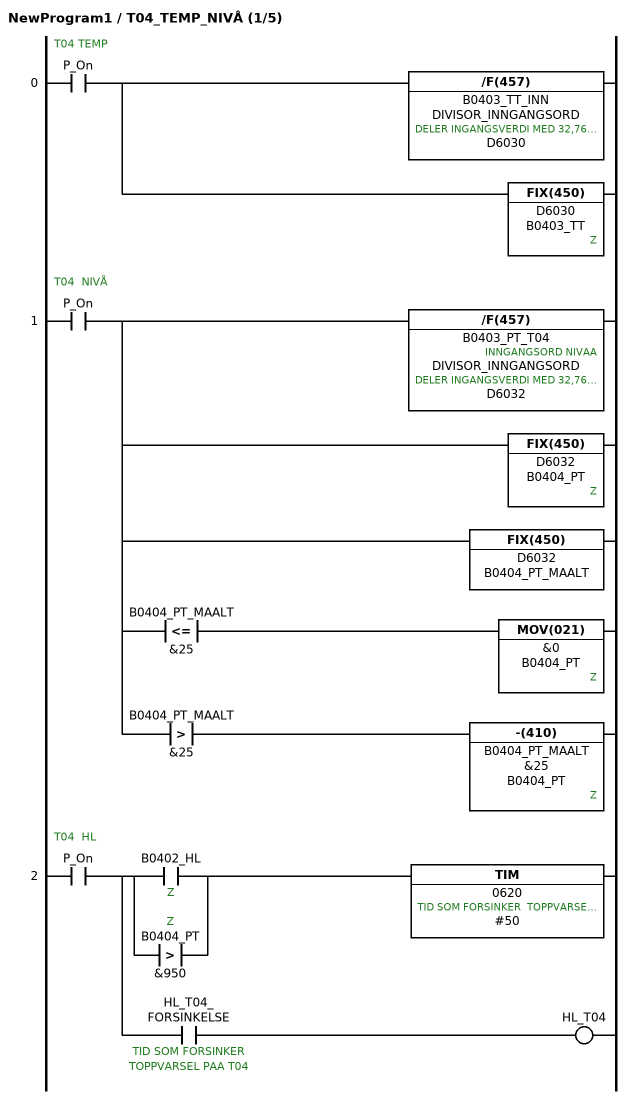
; [picture p912: NewProgram1 / T04_TEMP_NIVÅ, rungs 0-2]
; rung 0: T04 TEMP
LD P_On
/F(457) B0403_TT_INN DIVISOR_INNGANGSORD D6030  ; DELER INGANGSVERDI MED 32,760 FOR OMREGNING TIL 0-1000
FIX(450) D6030 B0403_TT  ; Z
; rung 1: T04  NIVÅ
LD P_On
OUT TR0
/F(457) B0403_PT_T04 DIVISOR_INNGANGSORD D6032  ; INNGANGSORD NIVAA, DELER INGANGSVERDI MED 32,760 FOR OMREGNING TIL 0-1000
FIX(450) D6032 B0404_PT  ; Z
FIX(450) D6032 B0404_PT_MAALT
AND<=(315) B0404_PT_MAALT &25
MOV(021) &0 B0404_PT  ; Z
LD TR0
AND>(320) B0404_PT_MAALT &25
-(410) B0404_PT_MAALT &25 B0404_PT  ; Z
; rung 2: T04  HL
LD P_On
OUT TR0
LD B0402_HL  ; Z
OR>(320) B0404_PT &950  ; Z
ANDLD
TIM 0620 #50  ; TID SOM FORSINKER  TOPPVARSEL PAA T04
LD TR0
AND HL_T04_FORSINKELSE  ; TID SOM FORSINKER  TOPPVARSEL PAA T04
OUT HL_T04

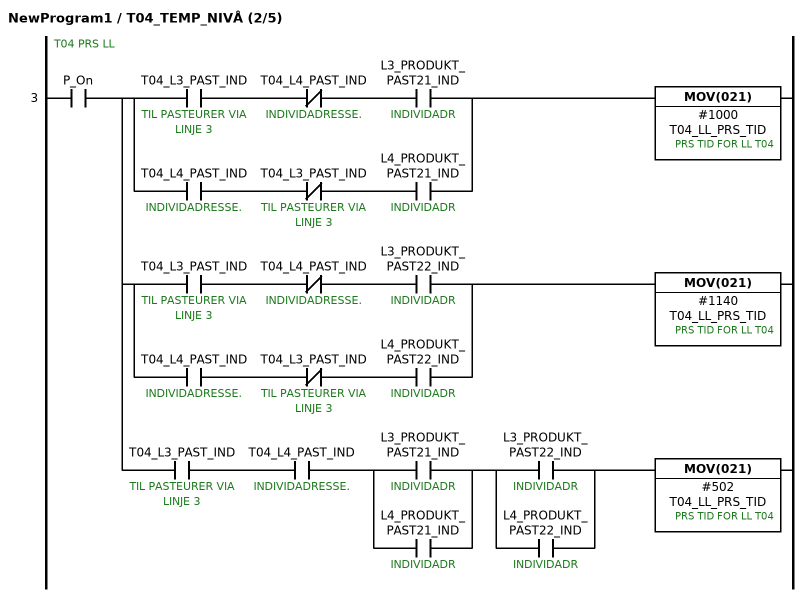
; rung 3: T04 PRS LL
LD P_On
OUT TR0
LD T04_L3_PAST_IND  ; TIL PASTEURER VIA LINJE 3
ANDNOT T04_L4_PAST_IND  ; INDIVIDADRESSE.
AND L3_PRODUKT_PAST21_IND  ; INDIVIDADR
LD T04_L4_PAST_IND  ; INDIVIDADRESSE.
ANDNOT T04_L3_PAST_IND  ; TIL PASTEURER VIA LINJE 3
AND L4_PRODUKT_PAST21_IND  ; INDIVIDADR
ORLD
ANDLD
MOV(021) #1000 T04_LL_PRS_TID  ; PRS TID FOR LL T04
LD TR0
LD T04_L3_PAST_IND  ; TIL PASTEURER VIA LINJE 3
ANDNOT T04_L4_PAST_IND  ; INDIVIDADRESSE.
AND L3_PRODUKT_PAST22_IND  ; INDIVIDADR
LD T04_L4_PAST_IND  ; INDIVIDADRESSE.
ANDNOT T04_L3_PAST_IND  ; TIL PASTEURER VIA LINJE 3
AND L4_PRODUKT_PAST22_IND  ; INDIVIDADR
ORLD
ANDLD
MOV(021) #1140 T04_LL_PRS_TID  ; PRS TID FOR LL T04
LD TR0
AND T04_L3_PAST_IND  ; TIL PASTEURER VIA LINJE 3
AND T04_L4_PAST_IND  ; INDIVIDADRESSE.
LD L3_PRODUKT_PAST21_IND  ; INDIVIDADR
OR L4_PRODUKT_PAST21_IND  ; INDIVIDADR
ANDLD
LD L3_PRODUKT_PAST22_IND  ; INDIVIDADR
OR L4_PRODUKT_PAST22_IND  ; INDIVIDADR
ANDLD
MOV(021) #502 T04_LL_PRS_TID  ; PRS TID FOR LL T04

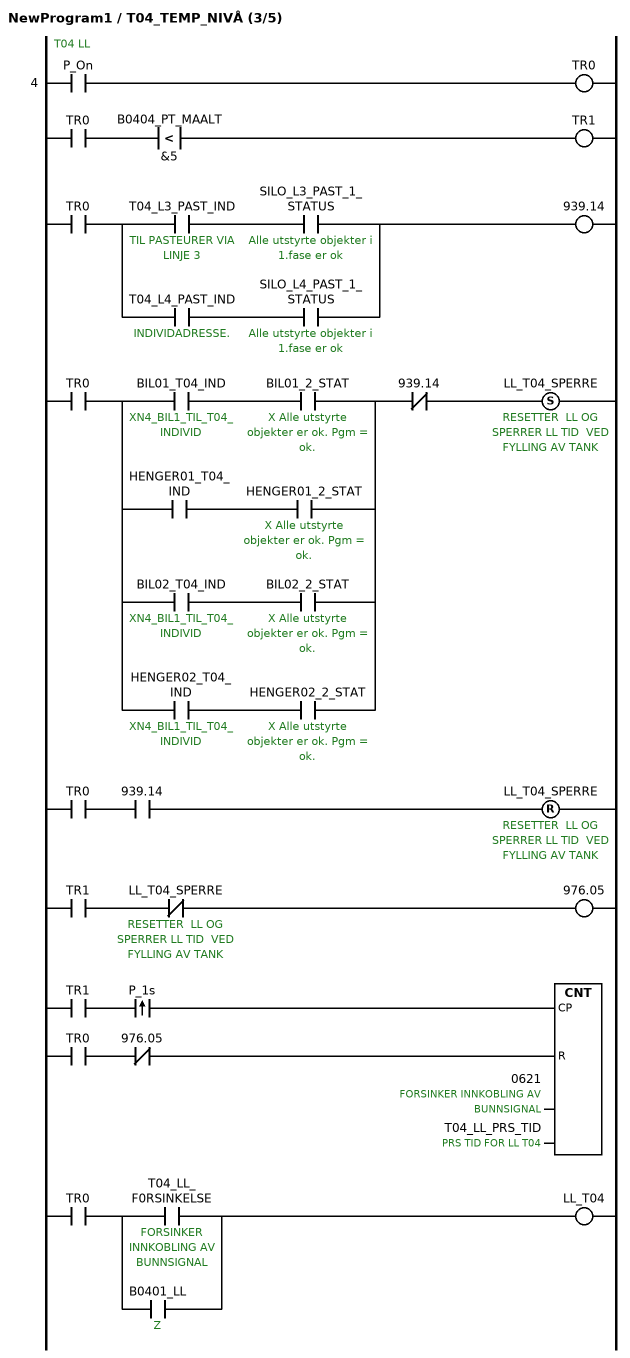
; rung 4: T04 LL
LD P_On
OUT TR0
LD T04_L3_PAST_IND  ; TIL PASTEURER VIA LINJE 3
AND SILO_L3_PAST_1_STATUS  ; Alle utstyrte objekter i 1.fase er ok
LD T04_L4_PAST_IND  ; INDIVIDADRESSE.
AND SILO_L4_PAST_1_STATUS  ; Alle utstyrte objekter i 1.fase er ok
ORLD
ANDLD
OUT 939.14
LD TR0
LD BIL01_T04_IND  ; XN4_BIL1_TIL_T04_INDIVID
AND BIL01_2_STAT  ; X Alle utstyrte objekter er ok. Pgm = ok.
LD HENGER01_T04_IND
AND HENGER01_2_STAT  ; X Alle utstyrte objekter er ok. Pgm = ok.
ORLD
LD BIL02_T04_IND  ; XN4_BIL1_TIL_T04_INDIVID
AND BIL02_2_STAT  ; X Alle utstyrte objekter er ok. Pgm = ok.
ORLD
LD HENGER02_T04_IND  ; XN4_BIL1_TIL_T04_INDIVID
AND HENGER02_2_STAT  ; X Alle utstyrte objekter er ok. Pgm = ok.
ORLD
ANDLD
ANDNOT 939.14
SET LL_T04_SPERRE  ; RESETTER  LL OG SPERRER LL TID  VED FYLLING AV TANK
LD TR0
AND 939.14
RSET LL_T04_SPERRE  ; RESETTER  LL OG SPERRER LL TID  VED FYLLING AV TANK
LD TR0
AND<(310) B0404_PT_MAALT &5
OUT TR1
ANDNOT LL_T04_SPERRE  ; RESETTER  LL OG SPERRER LL TID  VED FYLLING AV TANK
OUT 976.05
LD TR1
@AND P_1s
LD TR0
ANDNOT 976.05
CNT 0621 T04_LL_PRS_TID  ; PRS TID FOR LL T04, FORSINKER INNKOBLING AV BUNNSIGNAL
LD TR0
LD T04_LL_F0RSINKELSE  ; FORSINKER INNKOBLING AV BUNNSIGNAL
OR B0401_LL  ; Z
ANDLD
OUT LL_T04

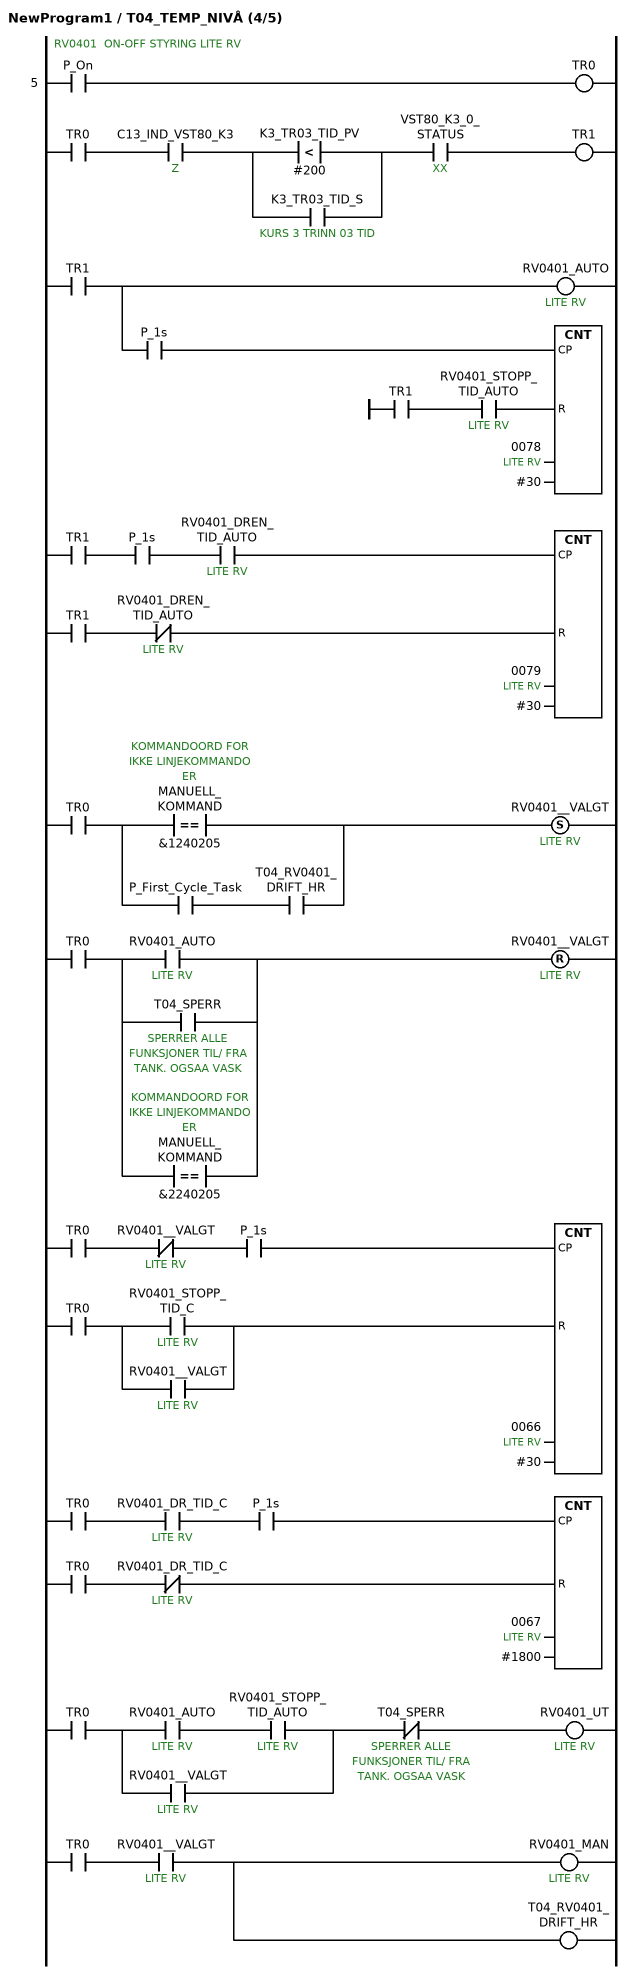
; rung 5: RV0401  ON-OFF STYRING LITE RV
LD P_On
OUT TR0
AND C13_IND_VST80_K3  ; Z
LD<(310) K3_TR03_TID_PV #200
OR K3_TR03_TID_S  ; KURS 3 TRINN 03 TID
ANDLD
AND VST80_K3_0_STATUS  ; XX
OUT TR1
OUT RV0401_AUTO  ; LITE RV
AND P_1s
LD TR1
AND RV0401_STOPP_TID_AUTO  ; LITE RV
CNT 0078 #30  ; LITE RV
LD TR1
AND P_1s
AND RV0401_DREN_TID_AUTO  ; LITE RV
LD TR1
ANDNOT RV0401_DREN_TID_AUTO  ; LITE RV
CNT 0079 #30  ; LITE RV
LD TR0
LD=L(301) MANUELL_KOMMAND &1240205  ; KOMMANDOORD FOR IKKE LINJEKOMMANDOER
LD P_First_Cycle_Task
AND T04_RV0401_DRIFT_HR
ORLD
ANDLD
SET RV0401__VALGT  ; LITE RV
LD TR0
LD RV0401_AUTO  ; LITE RV
OR T04_SPERR  ; SPERRER ALLE FUNKSJONER TIL/ FRA TANK. OGSAA VASK
OR=L(301) MANUELL_KOMMAND &2240205  ; KOMMANDOORD FOR IKKE LINJEKOMMANDOER
ANDLD
RSET RV0401__VALGT  ; LITE RV
LD TR0
ANDNOT RV0401__VALGT  ; LITE RV
AND P_1s
LD TR0
LD RV0401_STOPP_TID_C  ; LITE RV
OR RV0401__VALGT  ; LITE RV
ANDLD
CNT 0066 #30  ; LITE RV
LD TR0
AND RV0401_DR_TID_C  ; LITE RV
AND P_1s
LD TR0
ANDNOT RV0401_DR_TID_C  ; LITE RV
CNT 0067 #1800  ; LITE RV
LD TR0
LD RV0401_AUTO  ; LITE RV
AND RV0401_STOPP_TID_AUTO  ; LITE RV
OR RV0401__VALGT  ; LITE RV
ANDLD
ANDNOT T04_SPERR  ; SPERRER ALLE FUNKSJONER TIL/ FRA TANK. OGSAA VASK
OUT RV0401_UT  ; LITE RV
LD TR0
AND RV0401__VALGT  ; LITE RV
OUT RV0401_MAN  ; LITE RV
OUT T04_RV0401_DRIFT_HR

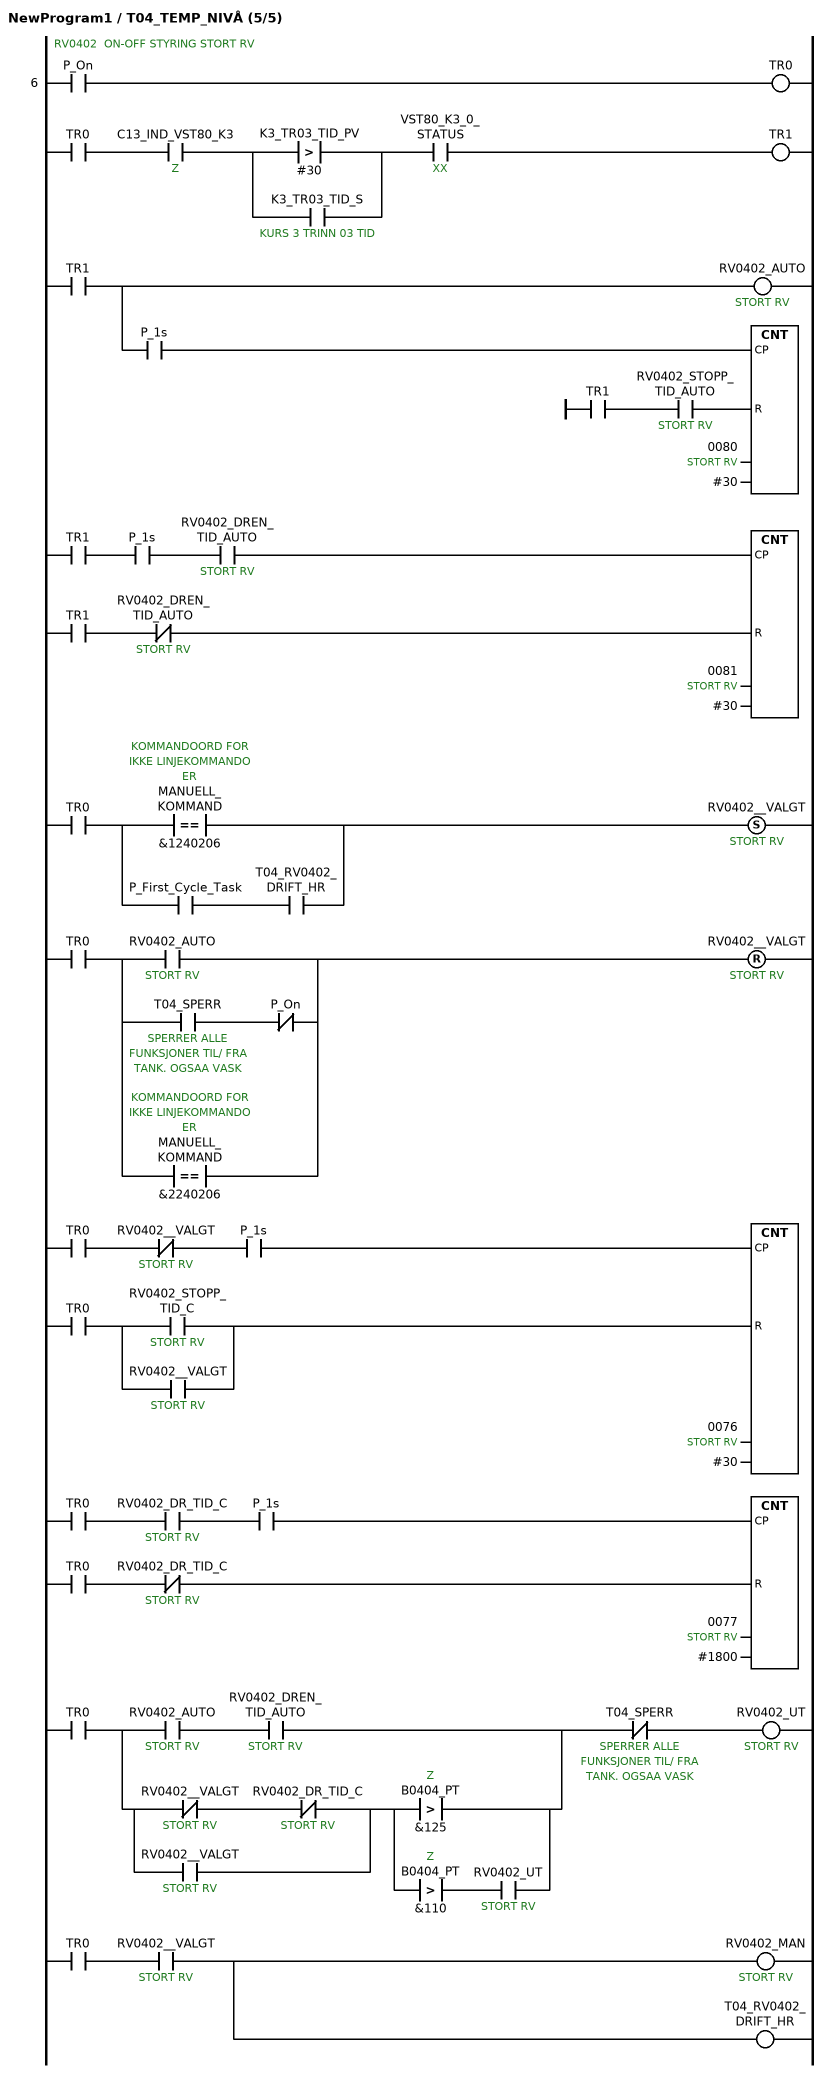
; rung 6: RV0402  ON-OFF STYRING STORT RV
LD P_On
OUT TR0
AND C13_IND_VST80_K3  ; Z
LD>(320) K3_TR03_TID_PV #30
OR K3_TR03_TID_S  ; KURS 3 TRINN 03 TID
ANDLD
AND VST80_K3_0_STATUS  ; XX
OUT TR1
OUT RV0402_AUTO  ; STORT RV
AND P_1s
LD TR1
AND RV0402_STOPP_TID_AUTO  ; STORT RV
CNT 0080 #30  ; STORT RV
LD TR1
AND P_1s
AND RV0402_DREN_TID_AUTO  ; STORT RV
LD TR1
ANDNOT RV0402_DREN_TID_AUTO  ; STORT RV
CNT 0081 #30  ; STORT RV
LD TR0
LD=L(301) MANUELL_KOMMAND &1240206  ; KOMMANDOORD FOR IKKE LINJEKOMMANDOER
LD P_First_Cycle_Task
AND T04_RV0402_DRIFT_HR
ORLD
ANDLD
SET RV0402__VALGT  ; STORT RV
LD TR0
LD RV0402_AUTO  ; STORT RV
LD T04_SPERR  ; SPERRER ALLE FUNKSJONER TIL/ FRA TANK. OGSAA VASK
ANDNOT P_On
ORLD
OR=L(301) MANUELL_KOMMAND &2240206  ; KOMMANDOORD FOR IKKE LINJEKOMMANDOER
ANDLD
RSET RV0402__VALGT  ; STORT RV
LD TR0
ANDNOT RV0402__VALGT  ; STORT RV
AND P_1s
LD TR0
LD RV0402_STOPP_TID_C  ; STORT RV
OR RV0402__VALGT  ; STORT RV
ANDLD
CNT 0076 #30  ; STORT RV
LD TR0
AND RV0402_DR_TID_C  ; STORT RV
AND P_1s
LD TR0
ANDNOT RV0402_DR_TID_C  ; STORT RV
CNT 0077 #1800  ; STORT RV
LD TR0
LD RV0402_AUTO  ; STORT RV
AND RV0402_DREN_TID_AUTO  ; STORT RV
LDNOT RV0402__VALGT  ; STORT RV
ANDNOT RV0402_DR_TID_C  ; STORT RV
OR RV0402__VALGT  ; STORT RV
LD>(320) B0404_PT &125  ; Z
LD>(320) B0404_PT &110  ; Z
AND RV0402_UT  ; STORT RV
ORLD
ANDLD
ORLD
ANDLD
ANDNOT T04_SPERR  ; SPERRER ALLE FUNKSJONER TIL/ FRA TANK. OGSAA VASK
OUT RV0402_UT  ; STORT RV
LD TR0
AND RV0402__VALGT  ; STORT RV
OUT RV0402_MAN  ; STORT RV
OUT T04_RV0402_DRIFT_HR
; rung 7: Ingen_kommentar_funnet

### Section T04_STATUS

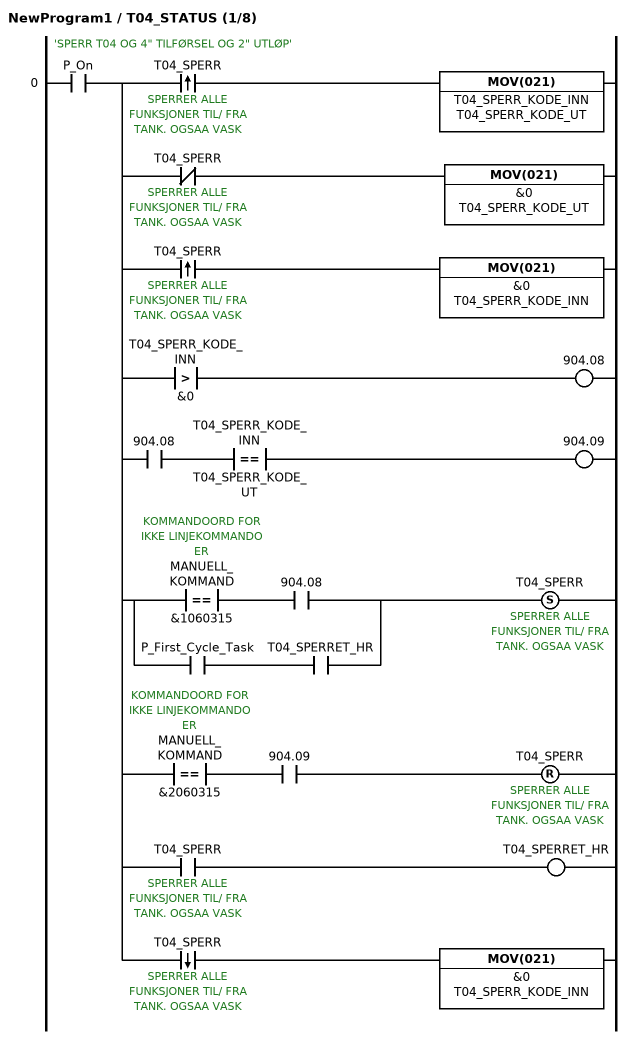
; rung 0: 'SPERR T04 OG 4" TILFØRSEL OG 2" UTLØP'
LD P_On
OUT TR0
@AND T04_SPERR  ; SPERRER ALLE FUNKSJONER TIL/ FRA TANK. OGSAA VASK
MOV(021) T04_SPERR_KODE_INN T04_SPERR_KODE_UT
LD TR0
ANDNOT T04_SPERR  ; SPERRER ALLE FUNKSJONER TIL/ FRA TANK. OGSAA VASK
MOV(021) &0 T04_SPERR_KODE_UT
LD TR0
@AND T04_SPERR  ; SPERRER ALLE FUNKSJONER TIL/ FRA TANK. OGSAA VASK
MOV(021) &0 T04_SPERR_KODE_INN
LD TR0
AND>(320) T04_SPERR_KODE_INN &0
OUT 904.08
LD TR0
AND 904.08
AND=(300) T04_SPERR_KODE_INN T04_SPERR_KODE_UT
OUT 904.09
LD TR0
LD=L(301) MANUELL_KOMMAND &1060315  ; KOMMANDOORD FOR IKKE LINJEKOMMANDOER
AND 904.08
LD P_First_Cycle_Task
AND T04_SPERRET_HR
ORLD
ANDLD
SET T04_SPERR  ; SPERRER ALLE FUNKSJONER TIL/ FRA TANK. OGSAA VASK
LD TR0
AND=L(301) MANUELL_KOMMAND &2060315  ; KOMMANDOORD FOR IKKE LINJEKOMMANDOER
AND 904.09
RSET T04_SPERR  ; SPERRER ALLE FUNKSJONER TIL/ FRA TANK. OGSAA VASK
LD TR0
AND T04_SPERR  ; SPERRER ALLE FUNKSJONER TIL/ FRA TANK. OGSAA VASK
OUT T04_SPERRET_HR
LD TR0
%AND T04_SPERR  ; SPERRER ALLE FUNKSJONER TIL/ FRA TANK. OGSAA VASK
MOV(021) &0 T04_SPERR_KODE_INN

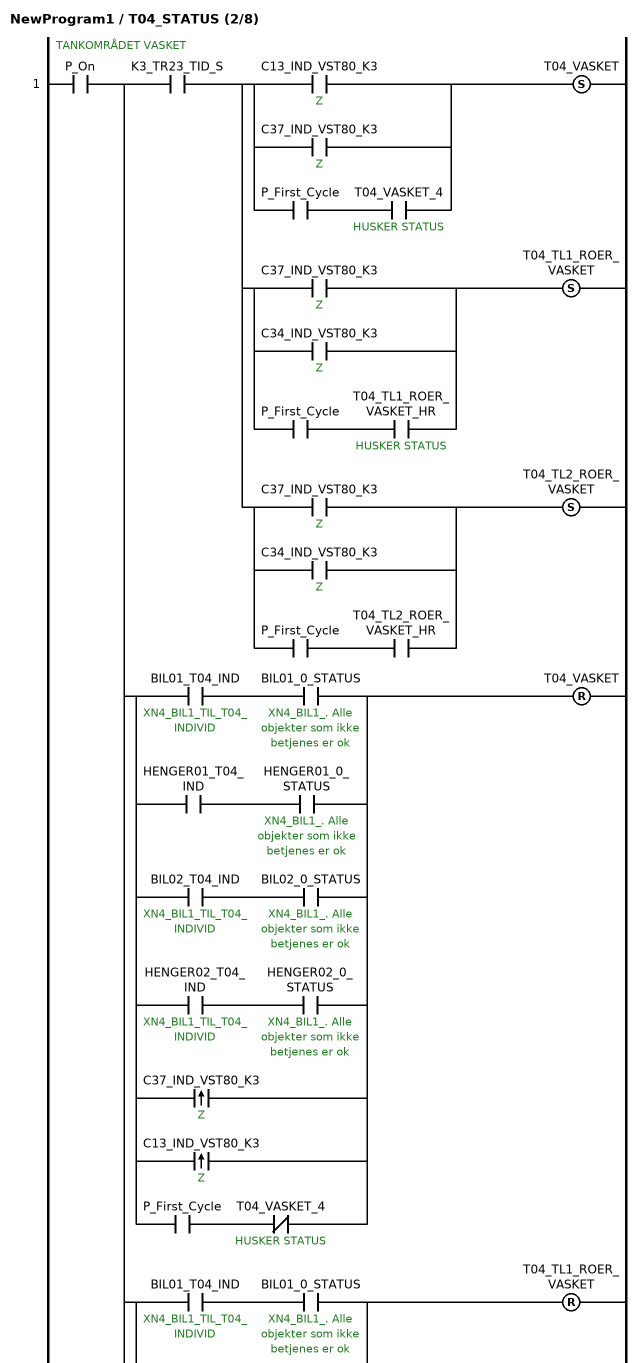

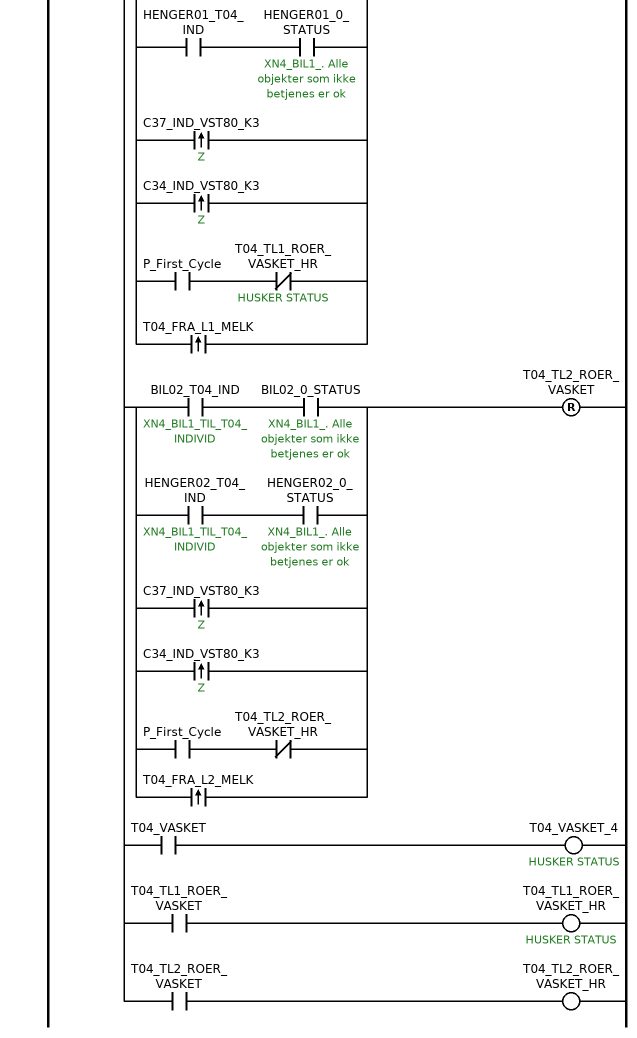
; rung 1: TANKOMRÅDET VASKET
LD P_On
OUT TR0
AND K3_TR23_TID_S
OUT TR1
LD C13_IND_VST80_K3  ; Z
OR C37_IND_VST80_K3  ; Z
LD P_First_Cycle
AND T04_VASKET_4  ; HUSKER STATUS
ORLD
ANDLD
SET T04_VASKET
LD TR1
LD C37_IND_VST80_K3  ; Z
OR C34_IND_VST80_K3  ; Z
LD P_First_Cycle
AND T04_TL1_ROER_VASKET_HR  ; HUSKER STATUS
ORLD
ANDLD
SET T04_TL1_ROER_VASKET
LD TR1
LD C37_IND_VST80_K3  ; Z
OR C34_IND_VST80_K3  ; Z
LD P_First_Cycle
AND T04_TL2_ROER_VASKET_HR
ORLD
ANDLD
SET T04_TL2_ROER_VASKET
LD TR0
LD BIL01_T04_IND  ; XN4_BIL1_TIL_T04_INDIVID
AND BIL01_0_STATUS  ; XN4_BIL1_. Alle objekter som ikke betjenes er ok
LD HENGER01_T04_IND
AND HENGER01_0_STATUS  ; XN4_BIL1_. Alle objekter som ikke betjenes er ok
ORLD
LD BIL02_T04_IND  ; XN4_BIL1_TIL_T04_INDIVID
AND BIL02_0_STATUS  ; XN4_BIL1_. Alle objekter som ikke betjenes er ok
ORLD
LD HENGER02_T04_IND  ; XN4_BIL1_TIL_T04_INDIVID
AND HENGER02_0_STATUS  ; XN4_BIL1_. Alle objekter som ikke betjenes er ok
ORLD
@OR C37_IND_VST80_K3  ; Z
@OR C13_IND_VST80_K3  ; Z
LD P_First_Cycle
ANDNOT T04_VASKET_4  ; HUSKER STATUS
ORLD
ANDLD
RSET T04_VASKET
LD TR0
LD BIL01_T04_IND  ; XN4_BIL1_TIL_T04_INDIVID
AND BIL01_0_STATUS  ; XN4_BIL1_. Alle objekter som ikke betjenes er ok
LD HENGER01_T04_IND
AND HENGER01_0_STATUS  ; XN4_BIL1_. Alle objekter som ikke betjenes er ok
ORLD
@OR C37_IND_VST80_K3  ; Z
@OR C34_IND_VST80_K3  ; Z
LD P_First_Cycle
ANDNOT T04_TL1_ROER_VASKET_HR  ; HUSKER STATUS
ORLD
@OR T04_FRA_L1_MELK
ANDLD
RSET T04_TL1_ROER_VASKET
LD TR0
LD BIL02_T04_IND  ; XN4_BIL1_TIL_T04_INDIVID
AND BIL02_0_STATUS  ; XN4_BIL1_. Alle objekter som ikke betjenes er ok
LD HENGER02_T04_IND  ; XN4_BIL1_TIL_T04_INDIVID
AND HENGER02_0_STATUS  ; XN4_BIL1_. Alle objekter som ikke betjenes er ok
ORLD
@OR C37_IND_VST80_K3  ; Z
@OR C34_IND_VST80_K3  ; Z
LD P_First_Cycle
ANDNOT T04_TL2_ROER_VASKET_HR
ORLD
@OR T04_FRA_L2_MELK
ANDLD
RSET T04_TL2_ROER_VASKET
LD TR0
AND T04_VASKET
OUT T04_VASKET_4  ; HUSKER STATUS
LD TR0
AND T04_TL1_ROER_VASKET
OUT T04_TL1_ROER_VASKET_HR  ; HUSKER STATUS
LD TR0
AND T04_TL2_ROER_VASKET
OUT T04_TL2_ROER_VASKET_HR

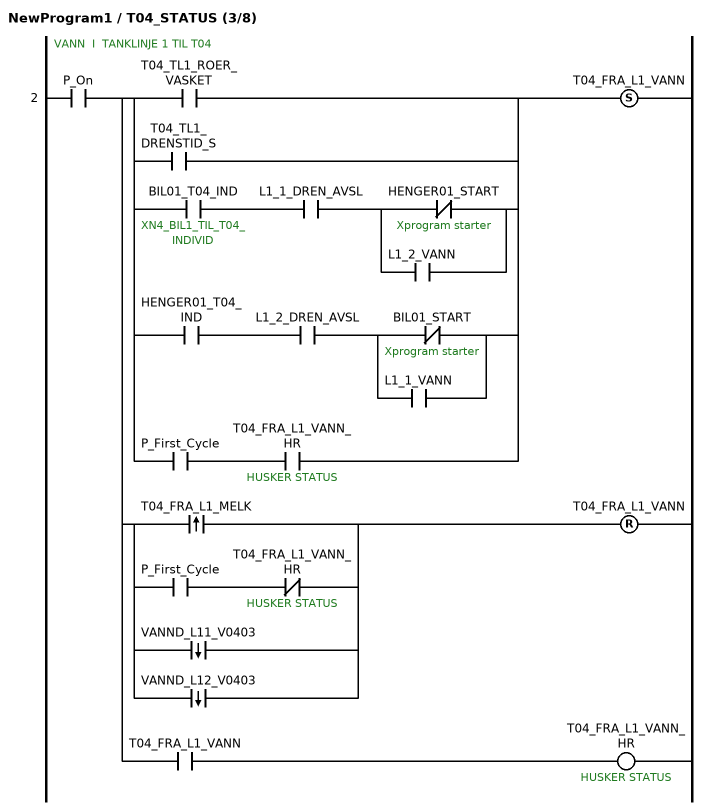
; rung 2: VANN  I  TANKLINJE 1 TIL T04
LD P_On
OUT TR0
LD T04_TL1_ROER_VASKET
OR T04_TL1_DRENSTID_S
LD BIL01_T04_IND  ; XN4_BIL1_TIL_T04_INDIVID
AND L1_1_DREN_AVSL
LDNOT HENGER01_START  ; Xprogram starter
OR L1_2_VANN
ANDLD
ORLD
LD HENGER01_T04_IND
AND L1_2_DREN_AVSL
LDNOT BIL01_START  ; Xprogram starter
OR L1_1_VANN
ANDLD
ORLD
LD P_First_Cycle
AND T04_FRA_L1_VANN_HR  ; HUSKER STATUS
ORLD
ANDLD
SET T04_FRA_L1_VANN
LD TR0
@LD T04_FRA_L1_MELK
LD P_First_Cycle
ANDNOT T04_FRA_L1_VANN_HR  ; HUSKER STATUS
ORLD
%OR VANND_L11_V0403
%OR VANND_L12_V0403
ANDLD
RSET T04_FRA_L1_VANN
LD TR0
AND T04_FRA_L1_VANN
OUT T04_FRA_L1_VANN_HR  ; HUSKER STATUS

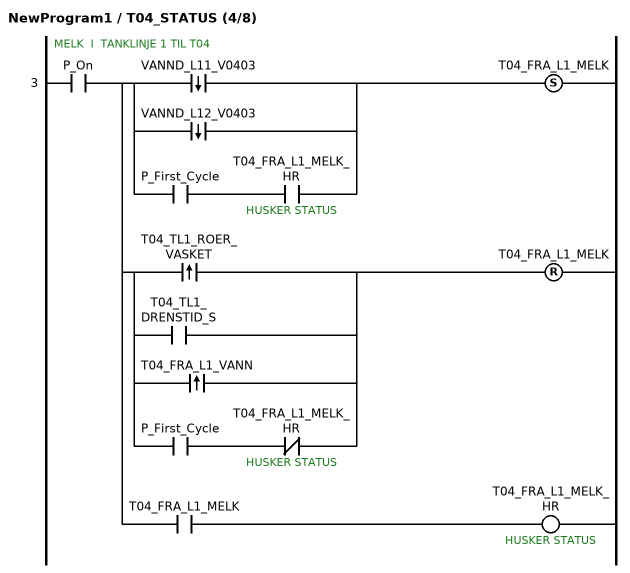
; rung 3: MELK  I  TANKLINJE 1 TIL T04
LD P_On
OUT TR0
%LD VANND_L11_V0403
%OR VANND_L12_V0403
LD P_First_Cycle
AND T04_FRA_L1_MELK_HR  ; HUSKER STATUS
ORLD
ANDLD
SET T04_FRA_L1_MELK
LD TR0
@LD T04_TL1_ROER_VASKET
OR T04_TL1_DRENSTID_S
@OR T04_FRA_L1_VANN
LD P_First_Cycle
ANDNOT T04_FRA_L1_MELK_HR  ; HUSKER STATUS
ORLD
ANDLD
RSET T04_FRA_L1_MELK
LD TR0
AND T04_FRA_L1_MELK
OUT T04_FRA_L1_MELK_HR  ; HUSKER STATUS

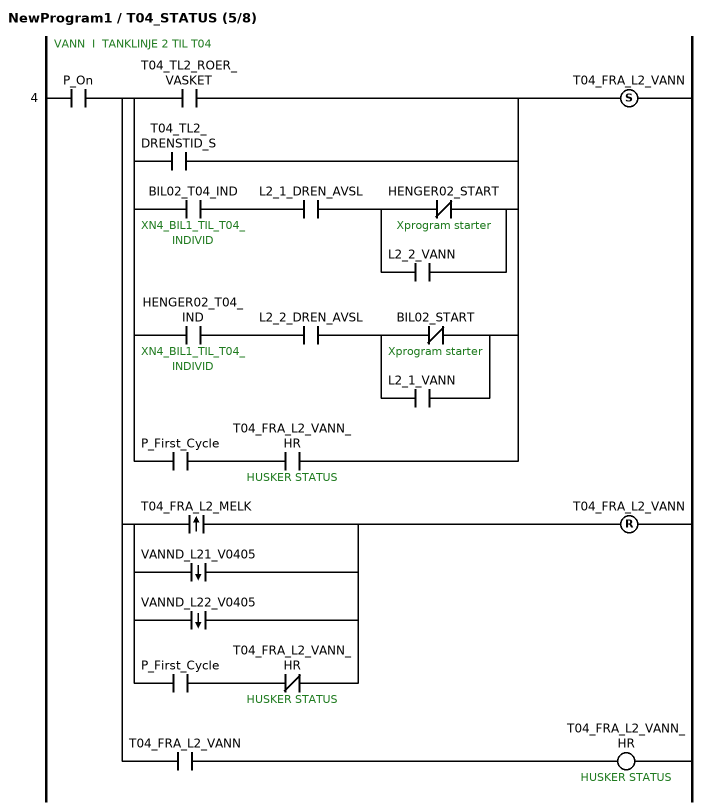
; rung 4: VANN  I  TANKLINJE 2 TIL T04
LD P_On
OUT TR0
LD T04_TL2_ROER_VASKET
OR T04_TL2_DRENSTID_S
LD BIL02_T04_IND  ; XN4_BIL1_TIL_T04_INDIVID
AND L2_1_DREN_AVSL
LDNOT HENGER02_START  ; Xprogram starter
OR L2_2_VANN
ANDLD
ORLD
LD HENGER02_T04_IND  ; XN4_BIL1_TIL_T04_INDIVID
AND L2_2_DREN_AVSL
LDNOT BIL02_START  ; Xprogram starter
OR L2_1_VANN
ANDLD
ORLD
LD P_First_Cycle
AND T04_FRA_L2_VANN_HR  ; HUSKER STATUS
ORLD
ANDLD
SET T04_FRA_L2_VANN
LD TR0
@LD T04_FRA_L2_MELK
%OR VANND_L21_V0405
%OR VANND_L22_V0405
LD P_First_Cycle
ANDNOT T04_FRA_L2_VANN_HR  ; HUSKER STATUS
ORLD
ANDLD
RSET T04_FRA_L2_VANN
LD TR0
AND T04_FRA_L2_VANN
OUT T04_FRA_L2_VANN_HR  ; HUSKER STATUS

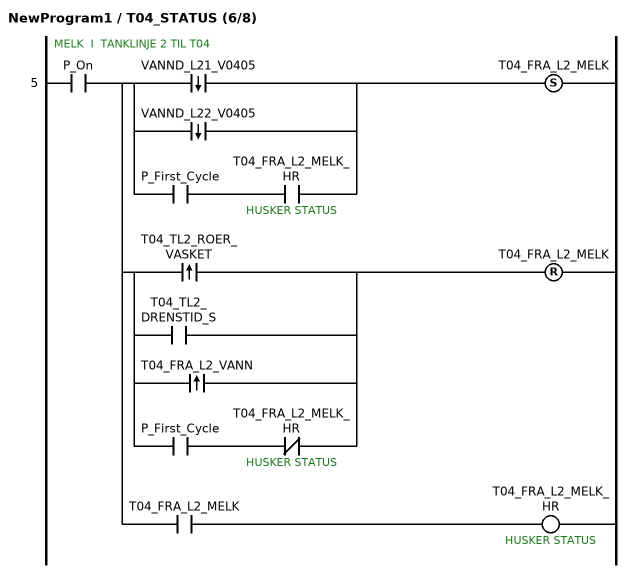
; rung 5: MELK  I  TANKLINJE 2 TIL T04
LD P_On
OUT TR0
%LD VANND_L21_V0405
%OR VANND_L22_V0405
LD P_First_Cycle
AND T04_FRA_L2_MELK_HR  ; HUSKER STATUS
ORLD
ANDLD
SET T04_FRA_L2_MELK
LD TR0
@LD T04_TL2_ROER_VASKET
OR T04_TL2_DRENSTID_S
@OR T04_FRA_L2_VANN
LD P_First_Cycle
ANDNOT T04_FRA_L2_MELK_HR  ; HUSKER STATUS
ORLD
ANDLD
RSET T04_FRA_L2_MELK
LD TR0
AND T04_FRA_L2_MELK
OUT T04_FRA_L2_MELK_HR  ; HUSKER STATUS

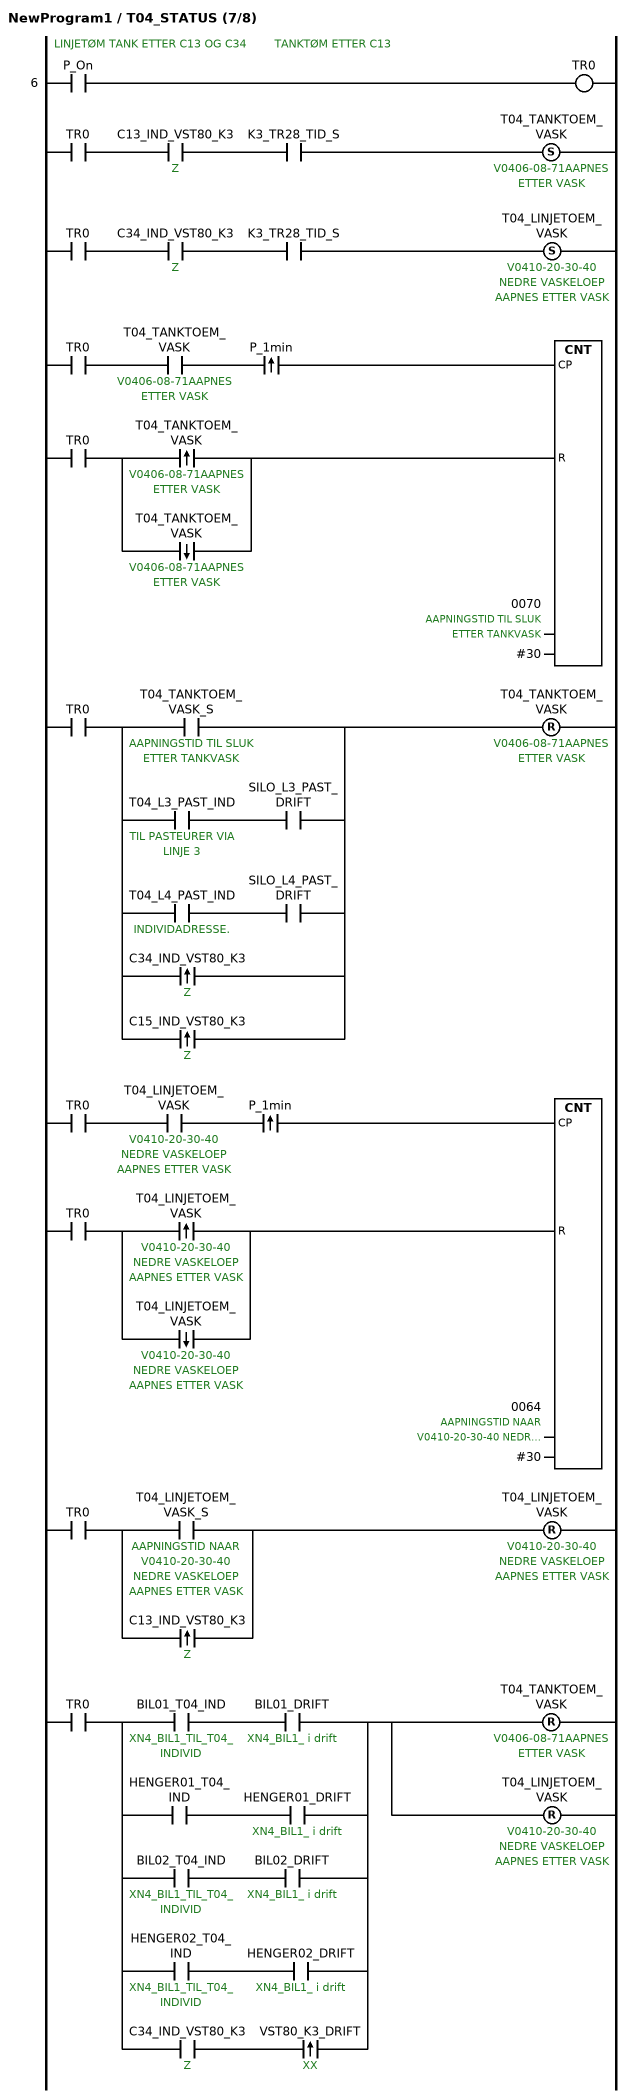
; rung 6: LINJETØM TANK ETTER C13 OG C34        TANKTØM ETTER C13
LD P_On
OUT TR0
AND C13_IND_VST80_K3  ; Z
AND K3_TR28_TID_S
SET T04_TANKTOEM_VASK  ; V0406-08-71AAPNES ETTER VASK
LD TR0
AND C34_IND_VST80_K3  ; Z
AND K3_TR28_TID_S
SET T04_LINJETOEM_VASK  ; V0410-20-30-40 NEDRE VASKELOEP AAPNES ETTER VASK
LD TR0
AND T04_TANKTOEM_VASK  ; V0406-08-71AAPNES ETTER VASK
@AND P_1min
LD TR0
@LD T04_TANKTOEM_VASK  ; V0406-08-71AAPNES ETTER VASK
%OR T04_TANKTOEM_VASK  ; V0406-08-71AAPNES ETTER VASK
ANDLD
CNT 0070 #30  ; AAPNINGSTID TIL SLUK ETTER TANKVASK
LD TR0
LD T04_TANKTOEM_VASK_S  ; AAPNINGSTID TIL SLUK ETTER TANKVASK
LD T04_L3_PAST_IND  ; TIL PASTEURER VIA LINJE 3
AND SILO_L3_PAST_DRIFT
ORLD
LD T04_L4_PAST_IND  ; INDIVIDADRESSE.
AND SILO_L4_PAST_DRIFT
ORLD
@OR C34_IND_VST80_K3  ; Z
@OR C15_IND_VST80_K3  ; Z
ANDLD
RSET T04_TANKTOEM_VASK  ; V0406-08-71AAPNES ETTER VASK
LD TR0
AND T04_LINJETOEM_VASK  ; V0410-20-30-40 NEDRE VASKELOEP AAPNES ETTER VASK
@AND P_1min
LD TR0
@LD T04_LINJETOEM_VASK  ; V0410-20-30-40 NEDRE VASKELOEP AAPNES ETTER VASK
%OR T04_LINJETOEM_VASK  ; V0410-20-30-40 NEDRE VASKELOEP AAPNES ETTER VASK
ANDLD
CNT 0064 #30  ; AAPNINGSTID NAAR V0410-20-30-40 NEDRE VASKELOEP AAPNES ETTER VASK
LD TR0
LD T04_LINJETOEM_VASK_S  ; AAPNINGSTID NAAR V0410-20-30-40 NEDRE VASKELOEP AAPNES ETTER VASK
@OR C13_IND_VST80_K3  ; Z
ANDLD
RSET T04_LINJETOEM_VASK  ; V0410-20-30-40 NEDRE VASKELOEP AAPNES ETTER VASK
LD TR0
LD BIL01_T04_IND  ; XN4_BIL1_TIL_T04_INDIVID
AND BIL01_DRIFT  ; XN4_BIL1_ i drift
LD HENGER01_T04_IND
AND HENGER01_DRIFT  ; XN4_BIL1_ i drift
ORLD
LD BIL02_T04_IND  ; XN4_BIL1_TIL_T04_INDIVID
AND BIL02_DRIFT  ; XN4_BIL1_ i drift
ORLD
LD HENGER02_T04_IND  ; XN4_BIL1_TIL_T04_INDIVID
AND HENGER02_DRIFT  ; XN4_BIL1_ i drift
ORLD
LD C34_IND_VST80_K3  ; Z
@AND VST80_K3_DRIFT  ; XX
ORLD
ANDLD
RSET T04_TANKTOEM_VASK  ; V0406-08-71AAPNES ETTER VASK
RSET T04_LINJETOEM_VASK  ; V0410-20-30-40 NEDRE VASKELOEP AAPNES ETTER VASK

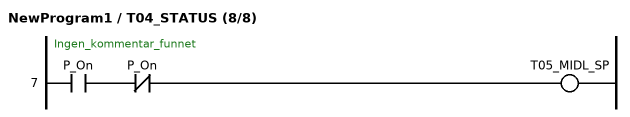
; rung 7: Ingen_kommentar_funnet
LD P_On
ANDNOT P_On
OUT T05_MIDL_SP
; rung 8: Ingen_kommentar_funnet

### Section T05_LOKALDREN

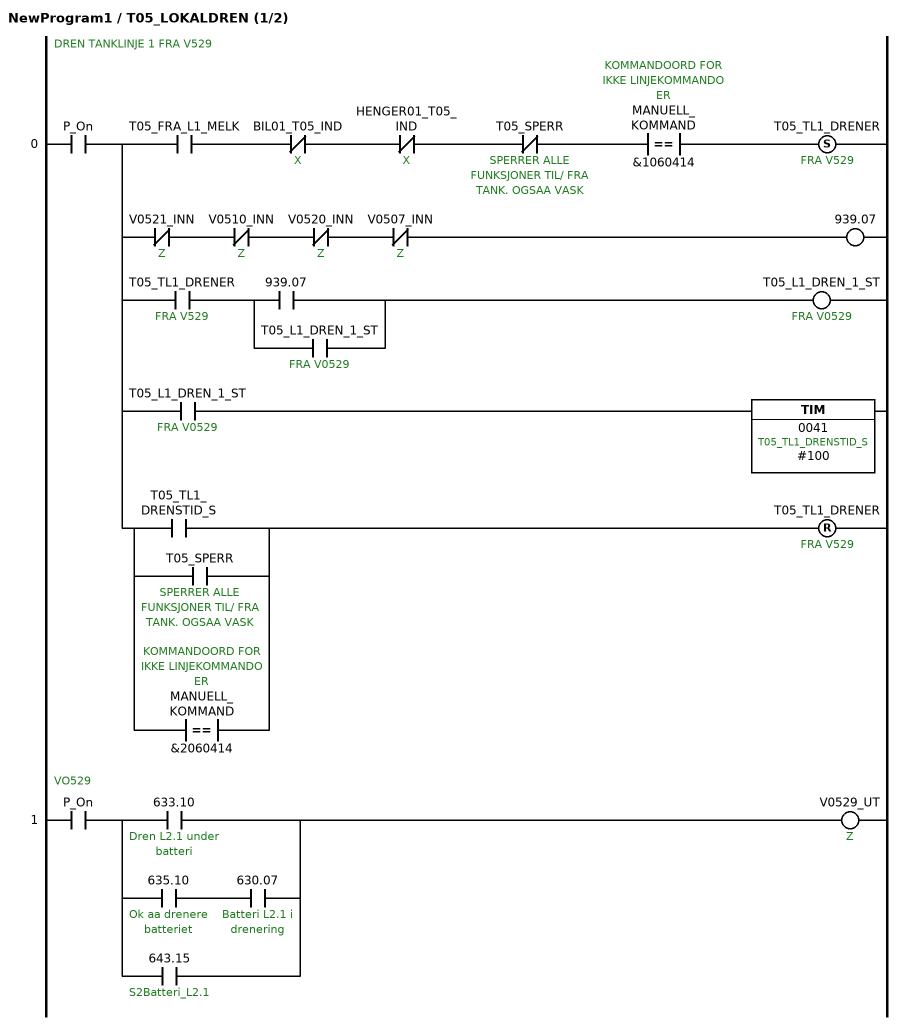
; rung 0: DREN TANKLINJE 1 FRA V529
LD P_On
OUT TR0
AND T05_FRA_L1_MELK
ANDNOT BIL01_T05_IND  ; X
ANDNOT HENGER01_T05_IND  ; X
ANDNOT T05_SPERR  ; SPERRER ALLE FUNKSJONER TIL/ FRA TANK. OGSAA VASK
AND=L(301) MANUELL_KOMMAND &1060414  ; KOMMANDOORD FOR IKKE LINJEKOMMANDOER
SET T05_TL1_DRENER  ; FRA V529
LD TR0
ANDNOT V0521_INN  ; Z
ANDNOT V0510_INN  ; Z
ANDNOT V0520_INN  ; Z
ANDNOT V0507_INN  ; Z
OUT 939.07
LD TR0
AND T05_TL1_DRENER  ; FRA V529
LD 939.07
OR T05_L1_DREN_1_ST  ; FRA V0529
ANDLD
OUT T05_L1_DREN_1_ST  ; FRA V0529
LD TR0
AND T05_L1_DREN_1_ST  ; FRA V0529
TIM 0041 #100  ; T05_TL1_DRENSTID_S
LD TR0
LD T05_TL1_DRENSTID_S
OR T05_SPERR  ; SPERRER ALLE FUNKSJONER TIL/ FRA TANK. OGSAA VASK
OR=L(301) MANUELL_KOMMAND &2060414  ; KOMMANDOORD FOR IKKE LINJEKOMMANDOER
ANDLD
RSET T05_TL1_DRENER  ; FRA V529
; rung 1: VO529
LD P_On
LD 633.10  ; Dren L2.1 under batteri
LD 635.10  ; Ok aa drenere batteriet
AND 630.07  ; Batteri L2.1 i drenering
ORLD
OR 643.15  ; S2Batteri_L2.1
ANDLD
OUT V0529_UT  ; Z

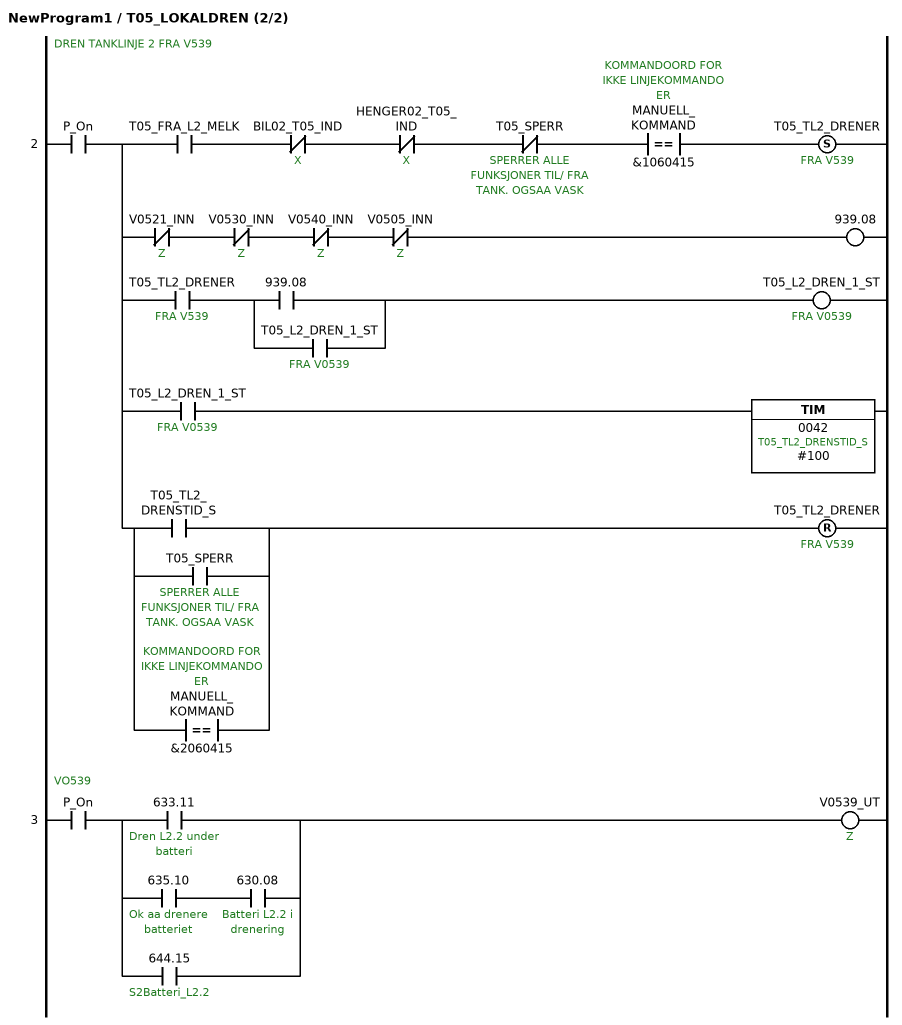
; rung 2: DREN TANKLINJE 2 FRA V539
LD P_On
OUT TR0
AND T05_FRA_L2_MELK
ANDNOT BIL02_T05_IND  ; X
ANDNOT HENGER02_T05_IND  ; X
ANDNOT T05_SPERR  ; SPERRER ALLE FUNKSJONER TIL/ FRA TANK. OGSAA VASK
AND=L(301) MANUELL_KOMMAND &1060415  ; KOMMANDOORD FOR IKKE LINJEKOMMANDOER
SET T05_TL2_DRENER  ; FRA V539
LD TR0
ANDNOT V0521_INN  ; Z
ANDNOT V0530_INN  ; Z
ANDNOT V0540_INN  ; Z
ANDNOT V0505_INN  ; Z
OUT 939.08
LD TR0
AND T05_TL2_DRENER  ; FRA V539
LD 939.08
OR T05_L2_DREN_1_ST  ; FRA V0539
ANDLD
OUT T05_L2_DREN_1_ST  ; FRA V0539
LD TR0
AND T05_L2_DREN_1_ST  ; FRA V0539
TIM 0042 #100  ; T05_TL2_DRENSTID_S
LD TR0
LD T05_TL2_DRENSTID_S
OR T05_SPERR  ; SPERRER ALLE FUNKSJONER TIL/ FRA TANK. OGSAA VASK
OR=L(301) MANUELL_KOMMAND &2060415  ; KOMMANDOORD FOR IKKE LINJEKOMMANDOER
ANDLD
RSET T05_TL2_DRENER  ; FRA V539
; rung 3: VO539
LD P_On
LD 633.11  ; Dren L2.2 under batteri
LD 635.10  ; Ok aa drenere batteriet
AND 630.08  ; Batteri L2.2 i drenering
ORLD
OR 644.15  ; S2Batteri_L2.2
ANDLD
OUT V0539_UT  ; Z
; rung 4: Ingen_kommentar_funnet

### Section T05_TEMP_NIVÅ

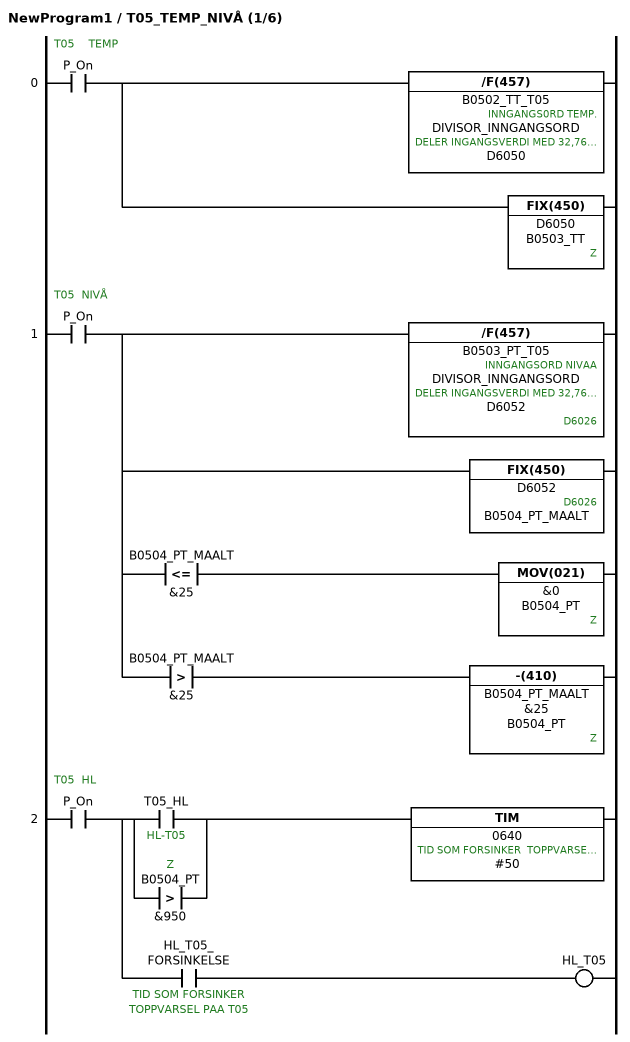
; rung 0: T05    TEMP
LD P_On
/F(457) B0502_TT_T05 DIVISOR_INNGANGSORD D6050  ; INNGANGS0RD TEMP., DELER INGANGSVERDI MED 32,760 FOR OMREGNING TIL 0-1000
FIX(450) D6050 B0503_TT  ; Z
; rung 1: T05  NIVÅ
LD P_On
OUT TR0
/F(457) B0503_PT_T05 DIVISOR_INNGANGSORD D6052  ; INNGANGSORD NIVAA, DELER INGANGSVERDI MED 32,760 FOR OMREGNING TIL 0-1000, D6026
FIX(450) D6052 B0504_PT_MAALT  ; D6026
AND<=(315) B0504_PT_MAALT &25
MOV(021) &0 B0504_PT  ; Z
LD TR0
AND>(320) B0504_PT_MAALT &25
-(410) B0504_PT_MAALT &25 B0504_PT  ; Z
; rung 2: T05  HL
LD P_On
OUT TR0
LD T05_HL  ; HL-T05
OR>(320) B0504_PT &950  ; Z
ANDLD
TIM 0640 #50  ; TID SOM FORSINKER  TOPPVARSEL PAA T05
LD TR0
AND HL_T05_FORSINKELSE  ; TID SOM FORSINKER  TOPPVARSEL PAA T05
OUT HL_T05

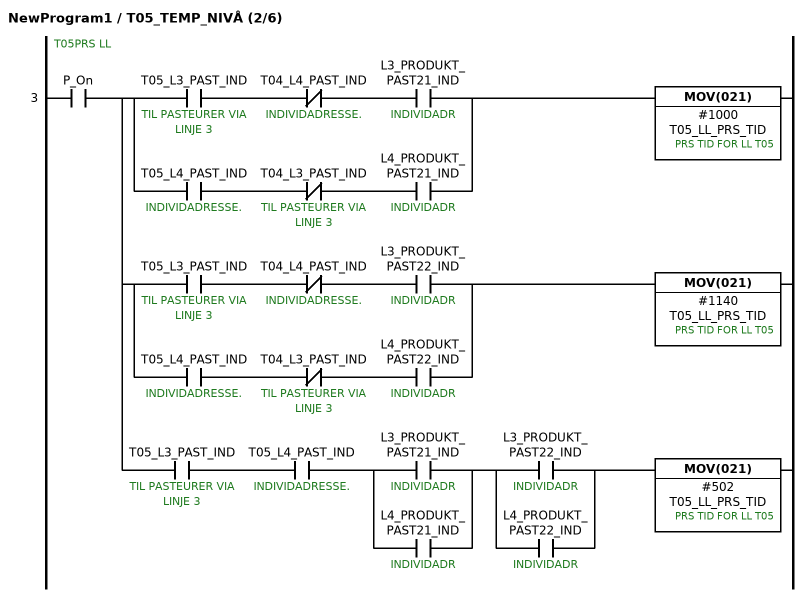
; rung 3: T05PRS LL
LD P_On
OUT TR0
LD T05_L3_PAST_IND  ; TIL PASTEURER VIA LINJE 3
ANDNOT T04_L4_PAST_IND  ; INDIVIDADRESSE.
AND L3_PRODUKT_PAST21_IND  ; INDIVIDADR
LD T05_L4_PAST_IND  ; INDIVIDADRESSE.
ANDNOT T04_L3_PAST_IND  ; TIL PASTEURER VIA LINJE 3
AND L4_PRODUKT_PAST21_IND  ; INDIVIDADR
ORLD
ANDLD
MOV(021) #1000 T05_LL_PRS_TID  ; PRS TID FOR LL T05
LD TR0
LD T05_L3_PAST_IND  ; TIL PASTEURER VIA LINJE 3
ANDNOT T04_L4_PAST_IND  ; INDIVIDADRESSE.
AND L3_PRODUKT_PAST22_IND  ; INDIVIDADR
LD T05_L4_PAST_IND  ; INDIVIDADRESSE.
ANDNOT T04_L3_PAST_IND  ; TIL PASTEURER VIA LINJE 3
AND L4_PRODUKT_PAST22_IND  ; INDIVIDADR
ORLD
ANDLD
MOV(021) #1140 T05_LL_PRS_TID  ; PRS TID FOR LL T05
LD TR0
AND T05_L3_PAST_IND  ; TIL PASTEURER VIA LINJE 3
AND T05_L4_PAST_IND  ; INDIVIDADRESSE.
LD L3_PRODUKT_PAST21_IND  ; INDIVIDADR
OR L4_PRODUKT_PAST21_IND  ; INDIVIDADR
ANDLD
LD L3_PRODUKT_PAST22_IND  ; INDIVIDADR
OR L4_PRODUKT_PAST22_IND  ; INDIVIDADR
ANDLD
MOV(021) #502 T05_LL_PRS_TID  ; PRS TID FOR LL T05

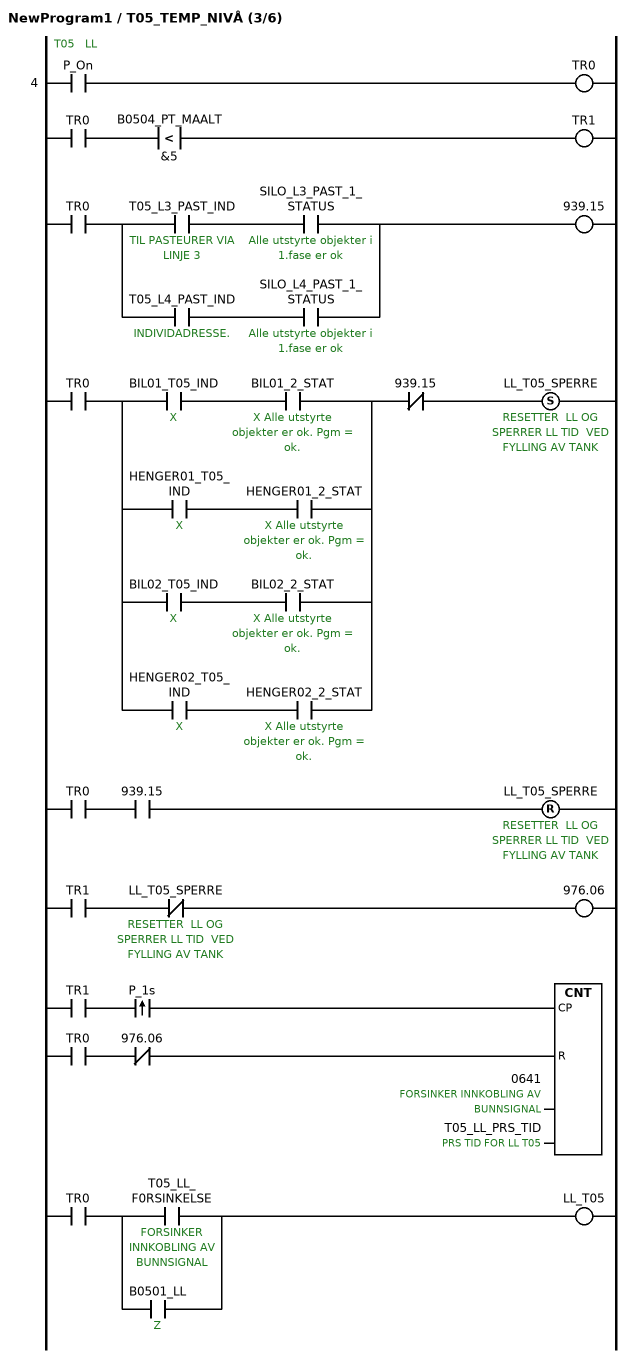
; rung 4: T05   LL
LD P_On
OUT TR0
LD T05_L3_PAST_IND  ; TIL PASTEURER VIA LINJE 3
AND SILO_L3_PAST_1_STATUS  ; Alle utstyrte objekter i 1.fase er ok
LD T05_L4_PAST_IND  ; INDIVIDADRESSE.
AND SILO_L4_PAST_1_STATUS  ; Alle utstyrte objekter i 1.fase er ok
ORLD
ANDLD
OUT 939.15
LD TR0
LD BIL01_T05_IND  ; X
AND BIL01_2_STAT  ; X Alle utstyrte objekter er ok. Pgm = ok.
LD HENGER01_T05_IND  ; X
AND HENGER01_2_STAT  ; X Alle utstyrte objekter er ok. Pgm = ok.
ORLD
LD BIL02_T05_IND  ; X
AND BIL02_2_STAT  ; X Alle utstyrte objekter er ok. Pgm = ok.
ORLD
LD HENGER02_T05_IND  ; X
AND HENGER02_2_STAT  ; X Alle utstyrte objekter er ok. Pgm = ok.
ORLD
ANDLD
ANDNOT 939.15
SET LL_T05_SPERRE  ; RESETTER  LL OG SPERRER LL TID  VED FYLLING AV TANK
LD TR0
AND 939.15
RSET LL_T05_SPERRE  ; RESETTER  LL OG SPERRER LL TID  VED FYLLING AV TANK
LD TR0
AND<(310) B0504_PT_MAALT &5
OUT TR1
ANDNOT LL_T05_SPERRE  ; RESETTER  LL OG SPERRER LL TID  VED FYLLING AV TANK
OUT 976.06
LD TR1
@AND P_1s
LD TR0
ANDNOT 976.06
CNT 0641 T05_LL_PRS_TID  ; PRS TID FOR LL T05, FORSINKER INNKOBLING AV BUNNSIGNAL
LD TR0
LD T05_LL_F0RSINKELSE  ; FORSINKER INNKOBLING AV BUNNSIGNAL
OR B0501_LL  ; Z
ANDLD
OUT LL_T05

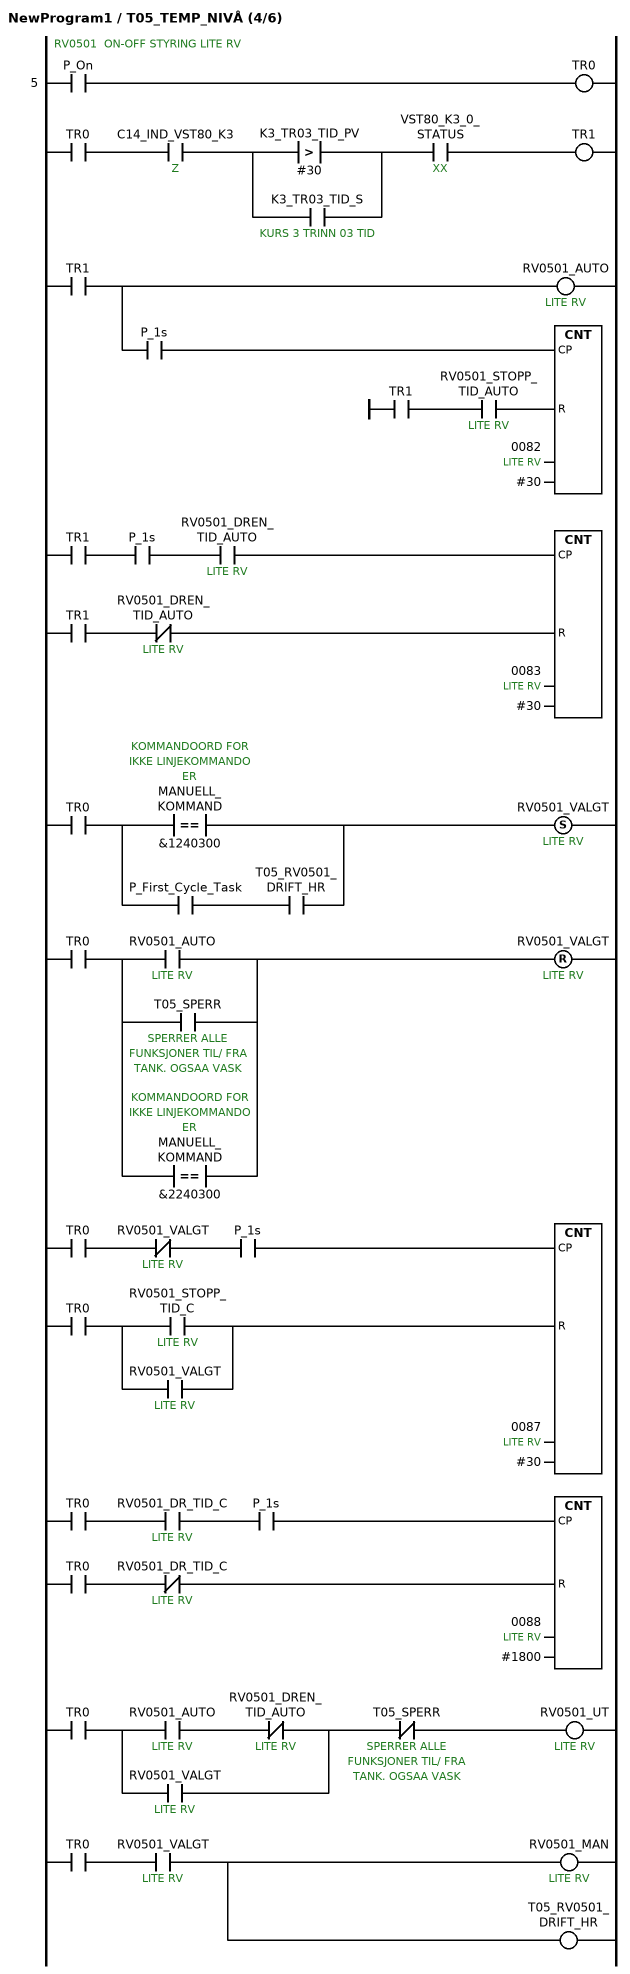
; rung 5: RV0501  ON-OFF STYRING LITE RV
LD P_On
OUT TR0
AND C14_IND_VST80_K3  ; Z
LD>(320) K3_TR03_TID_PV #30
OR K3_TR03_TID_S  ; KURS 3 TRINN 03 TID
ANDLD
AND VST80_K3_0_STATUS  ; XX
OUT TR1
OUT RV0501_AUTO  ; LITE RV
AND P_1s
LD TR1
AND RV0501_STOPP_TID_AUTO  ; LITE RV
CNT 0082 #30  ; LITE RV
LD TR1
AND P_1s
AND RV0501_DREN_TID_AUTO  ; LITE RV
LD TR1
ANDNOT RV0501_DREN_TID_AUTO  ; LITE RV
CNT 0083 #30  ; LITE RV
LD TR0
LD=L(301) MANUELL_KOMMAND &1240300  ; KOMMANDOORD FOR IKKE LINJEKOMMANDOER
LD P_First_Cycle_Task
AND T05_RV0501_DRIFT_HR
ORLD
ANDLD
SET RV0501_VALGT  ; LITE RV
LD TR0
LD RV0501_AUTO  ; LITE RV
OR T05_SPERR  ; SPERRER ALLE FUNKSJONER TIL/ FRA TANK. OGSAA VASK
OR=L(301) MANUELL_KOMMAND &2240300  ; KOMMANDOORD FOR IKKE LINJEKOMMANDOER
ANDLD
RSET RV0501_VALGT  ; LITE RV
LD TR0
ANDNOT RV0501_VALGT  ; LITE RV
AND P_1s
LD TR0
LD RV0501_STOPP_TID_C  ; LITE RV
OR RV0501_VALGT  ; LITE RV
ANDLD
CNT 0087 #30  ; LITE RV
LD TR0
AND RV0501_DR_TID_C  ; LITE RV
AND P_1s
LD TR0
ANDNOT RV0501_DR_TID_C  ; LITE RV
CNT 0088 #1800  ; LITE RV
LD TR0
LD RV0501_AUTO  ; LITE RV
ANDNOT RV0501_DREN_TID_AUTO  ; LITE RV
OR RV0501_VALGT  ; LITE RV
ANDLD
ANDNOT T05_SPERR  ; SPERRER ALLE FUNKSJONER TIL/ FRA TANK. OGSAA VASK
OUT RV0501_UT  ; LITE RV
LD TR0
AND RV0501_VALGT  ; LITE RV
OUT RV0501_MAN  ; LITE RV
OUT T05_RV0501_DRIFT_HR

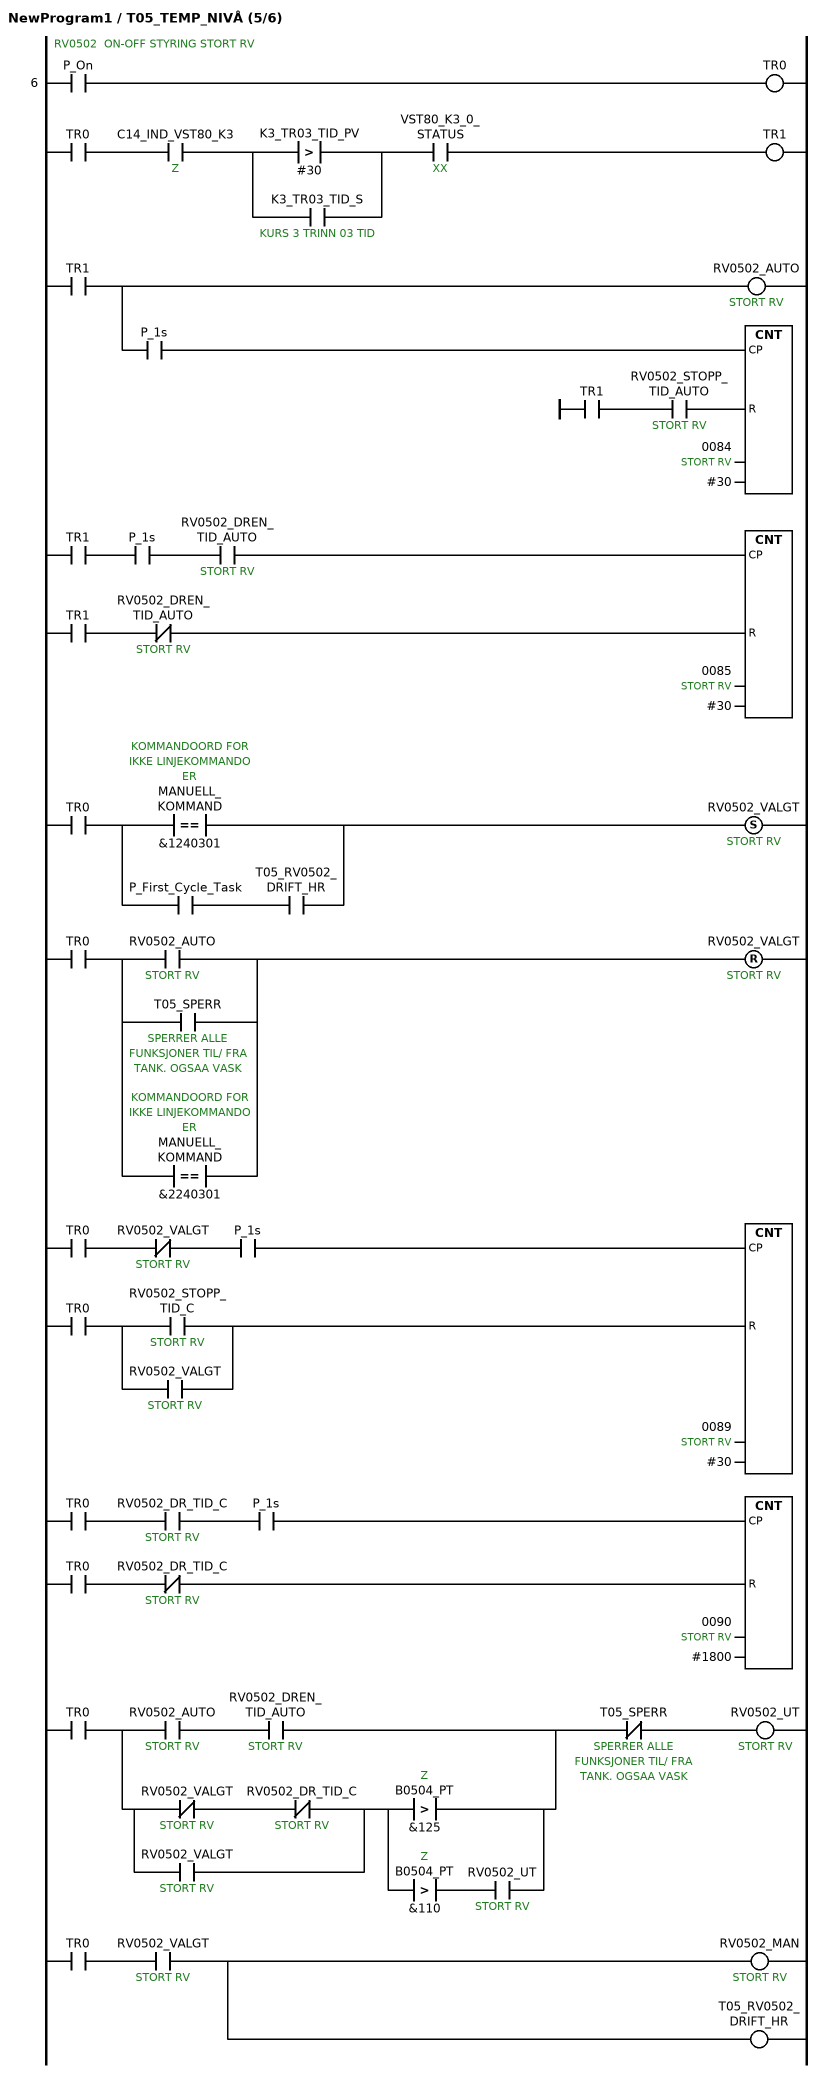
; rung 6: RV0502  ON-OFF STYRING STORT RV
LD P_On
OUT TR0
AND C14_IND_VST80_K3  ; Z
LD>(320) K3_TR03_TID_PV #30
OR K3_TR03_TID_S  ; KURS 3 TRINN 03 TID
ANDLD
AND VST80_K3_0_STATUS  ; XX
OUT TR1
OUT RV0502_AUTO  ; STORT RV
AND P_1s
LD TR1
AND RV0502_STOPP_TID_AUTO  ; STORT RV
CNT 0084 #30  ; STORT RV
LD TR1
AND P_1s
AND RV0502_DREN_TID_AUTO  ; STORT RV
LD TR1
ANDNOT RV0502_DREN_TID_AUTO  ; STORT RV
CNT 0085 #30  ; STORT RV
LD TR0
LD=L(301) MANUELL_KOMMAND &1240301  ; KOMMANDOORD FOR IKKE LINJEKOMMANDOER
LD P_First_Cycle_Task
AND T05_RV0502_DRIFT_HR
ORLD
ANDLD
SET RV0502_VALGT  ; STORT RV
LD TR0
LD RV0502_AUTO  ; STORT RV
OR T05_SPERR  ; SPERRER ALLE FUNKSJONER TIL/ FRA TANK. OGSAA VASK
OR=L(301) MANUELL_KOMMAND &2240301  ; KOMMANDOORD FOR IKKE LINJEKOMMANDOER
ANDLD
RSET RV0502_VALGT  ; STORT RV
LD TR0
ANDNOT RV0502_VALGT  ; STORT RV
AND P_1s
LD TR0
LD RV0502_STOPP_TID_C  ; STORT RV
OR RV0502_VALGT  ; STORT RV
ANDLD
CNT 0089 #30  ; STORT RV
LD TR0
AND RV0502_DR_TID_C  ; STORT RV
AND P_1s
LD TR0
ANDNOT RV0502_DR_TID_C  ; STORT RV
CNT 0090 #1800  ; STORT RV
LD TR0
LD RV0502_AUTO  ; STORT RV
AND RV0502_DREN_TID_AUTO  ; STORT RV
LDNOT RV0502_VALGT  ; STORT RV
ANDNOT RV0502_DR_TID_C  ; STORT RV
OR RV0502_VALGT  ; STORT RV
LD>(320) B0504_PT &125  ; Z
LD>(320) B0504_PT &110  ; Z
AND RV0502_UT  ; STORT RV
ORLD
ANDLD
ORLD
ANDLD
ANDNOT T05_SPERR  ; SPERRER ALLE FUNKSJONER TIL/ FRA TANK. OGSAA VASK
OUT RV0502_UT  ; STORT RV
LD TR0
AND RV0502_VALGT  ; STORT RV
OUT RV0502_MAN  ; STORT RV
OUT T05_RV0502_DRIFT_HR

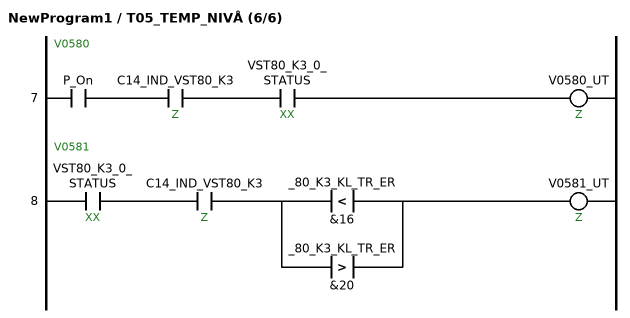
; rung 7: V0580
LD P_On
AND C14_IND_VST80_K3  ; Z
AND VST80_K3_0_STATUS  ; XX
OUT V0580_UT  ; Z
; rung 8: V0581
LD VST80_K3_0_STATUS  ; XX
AND C14_IND_VST80_K3  ; Z
LD<(310) _80_K3_KL_TR_ER &16
OR>(320) _80_K3_KL_TR_ER &20
ANDLD
OUT V0581_UT  ; Z
; rung 9: Ingen_kommentar_funnet

### Section T05_STATUS

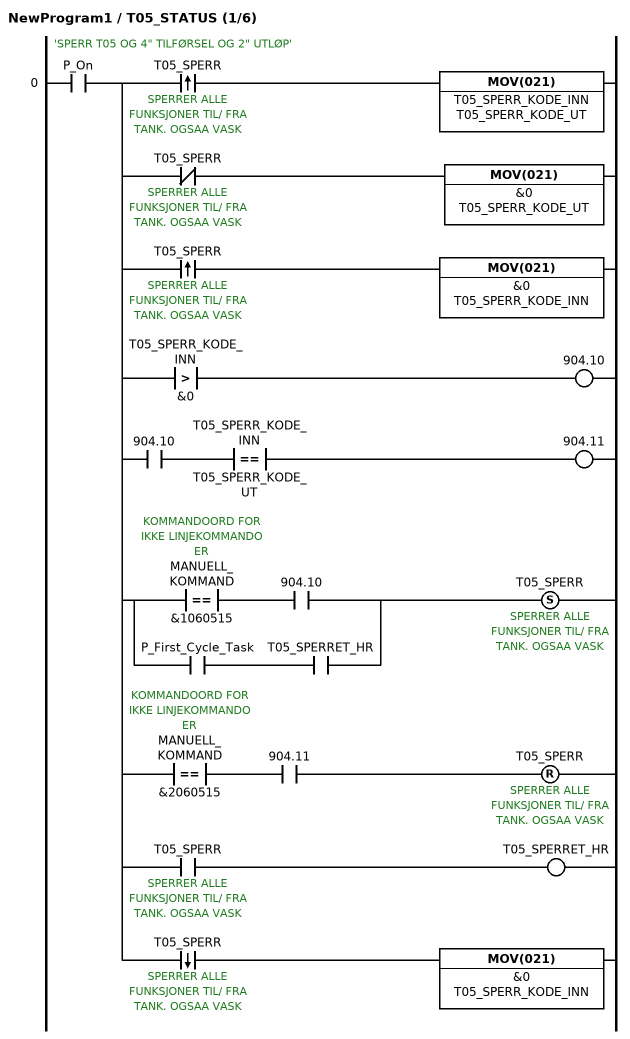
; rung 0: 'SPERR T05 OG 4" TILFØRSEL OG 2" UTLØP'
LD P_On
OUT TR0
@AND T05_SPERR  ; SPERRER ALLE FUNKSJONER TIL/ FRA TANK. OGSAA VASK
MOV(021) T05_SPERR_KODE_INN T05_SPERR_KODE_UT
LD TR0
ANDNOT T05_SPERR  ; SPERRER ALLE FUNKSJONER TIL/ FRA TANK. OGSAA VASK
MOV(021) &0 T05_SPERR_KODE_UT
LD TR0
@AND T05_SPERR  ; SPERRER ALLE FUNKSJONER TIL/ FRA TANK. OGSAA VASK
MOV(021) &0 T05_SPERR_KODE_INN
LD TR0
AND>(320) T05_SPERR_KODE_INN &0
OUT 904.10
LD TR0
AND 904.10
AND=(300) T05_SPERR_KODE_INN T05_SPERR_KODE_UT
OUT 904.11
LD TR0
LD=L(301) MANUELL_KOMMAND &1060515  ; KOMMANDOORD FOR IKKE LINJEKOMMANDOER
AND 904.10
LD P_First_Cycle_Task
AND T05_SPERRET_HR
ORLD
ANDLD
SET T05_SPERR  ; SPERRER ALLE FUNKSJONER TIL/ FRA TANK. OGSAA VASK
LD TR0
AND=L(301) MANUELL_KOMMAND &2060515  ; KOMMANDOORD FOR IKKE LINJEKOMMANDOER
AND 904.11
RSET T05_SPERR  ; SPERRER ALLE FUNKSJONER TIL/ FRA TANK. OGSAA VASK
LD TR0
AND T05_SPERR  ; SPERRER ALLE FUNKSJONER TIL/ FRA TANK. OGSAA VASK
OUT T05_SPERRET_HR
LD TR0
%AND T05_SPERR  ; SPERRER ALLE FUNKSJONER TIL/ FRA TANK. OGSAA VASK
MOV(021) &0 T05_SPERR_KODE_INN

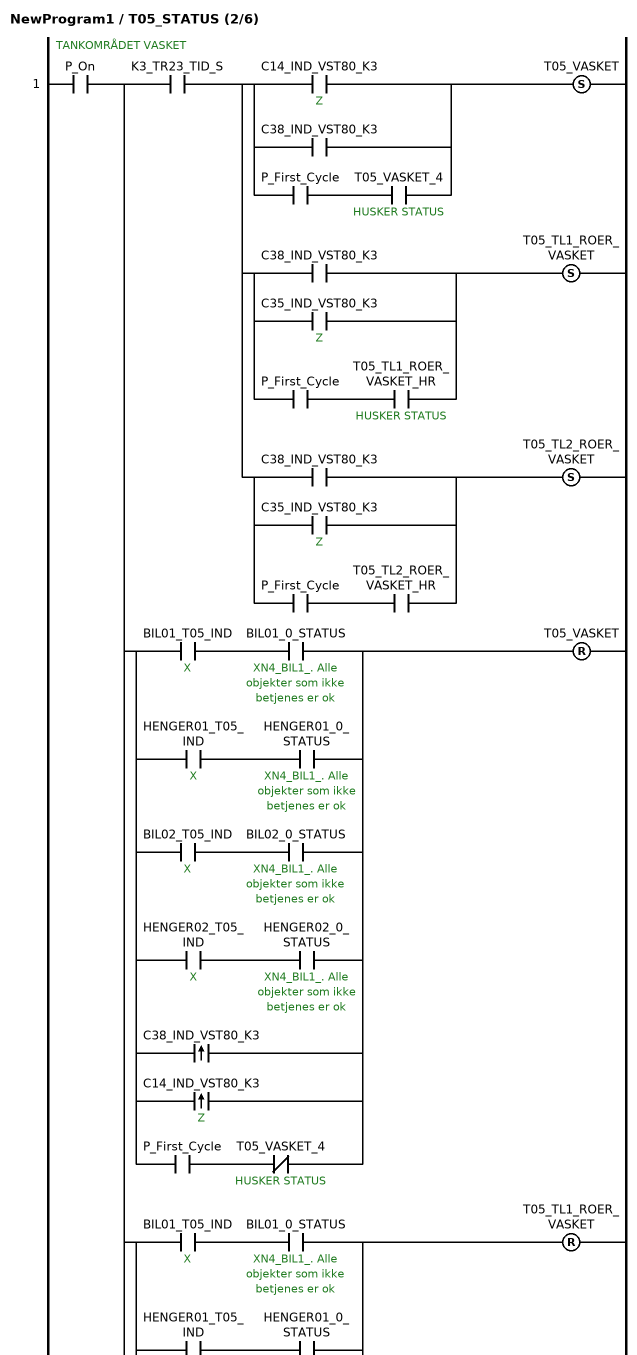

